Fanuc KAREL source: ko00093.KL

-- PROVISIONAL review KL for V1013-1; original PC SHA256 a43cb2992e61e449017f93ef57da8f078cae34ba91e91a32e7a0e0416b094595
-- Incomplete behavior may be omitted. Consult companion uncertainty JSON. Do not deploy.
PROGRAM KO00093
%NOLOCKGROUP
BEGIN
  -- UNRESOLVED_PC offsets 5-12; opcodes 9D,23
  -- UNRESOLVED_PC offsets 17-69; opcodes 27,27,49,7E,AD,27,49,7E,AD,22,31,7E,4A
  -- UNRESOLVED_PC offsets 74-78; opcodes 7F
END KO00093
